// TIA Portal V16 export
// export: Created 2024-09-05T17:39:11.3590484Z, ExportSetting WithDefaults, DisplayName Totally Integrated Automation Portal, DisplayVersion V16 Update 6, DisplayName TIA Portal Version Control Interface, DisplayVersion V16 Update 2, DisplayName TIA Portal Openness, DisplayVersion V16 Update 6, DisplayName STEP 7 Professional, DisplayVersion V16 Update 6, DisplayName STEP 7 Safety, DisplayVersion V16, DisplayName WinCC Advanced, DisplayVersion V16 Update 6
DATA_BLOCK "DiagnosticMain_DB"   // DB7
VERSION : 0.1
// stored: AutoNumber true, DBAccessibleFromOPCUA true, InstanceOfName DiagnosticMain, InstanceOfType FB
"DiagnosticMain"
   // VAR
   //    i : Int := 201;
   //    index : Int := 20;
   //    state : Int := 1;
   // END_VAR
BEGIN
END_DATA_BLOCK
